SUBAPPLICATION SubApp_PC_B (* Geraet B (Station 12, 192.168.1.12): identisch zu Training_10 (2x AX_SUBSCRIBE_1 -> ILOCK_SWITCH_PROTECT_AX -> 2x logiBUS_QXA), zusaetzlich schreibt der tatsaechlich erreichte Zustand (UP_OUT/DOWN_OUT NACH Arbitrierung/Schutzzeit) per AX_SPLIT_2 + AX_CLIENT_1_0 zurueck an Geraet A fuer die GreenWhiteBackground-Anzeige - analog zum Vorbild SoftKeySR_PC_A_OPC.SUB (dort State-Write von B nach A, hier gleiches Prinzip). *)
  (* Standard: 61499-2; Description: Copyright (c) 2026 Meisterschulen am Ostbahnhof This program and the accompanying materials are made available under the terms of the Eclipse Public License 2.0 which is available at https://www.eclipse.org/legal/epl-2.0/ SPDX-License-Identifier: EPL-2.0 *)
  (* Version 1.0, 2026-09-05, Franz Höpfinger, Meisterschulen am Ostbahnhof, initial API and implementation and/or initial documentation *)
  PACKAGE subapp::Training_11_OPC_UA_RES;
  IMPORT VV::const::OPC_UA::myOpcUaAddresses::SW1_UP_LOCAL_READ;
  IMPORT VV::const::OPC_UA::myOpcUaAddresses::SW1_DOWN_LOCAL_READ;
  IMPORT VV::const::OPC_UA::myOpcUaAddresses::SW1_UP_STATE_REMOTE_WRITE;
  IMPORT VV::const::OPC_UA::myOpcUaAddresses::SW1_DOWN_STATE_REMOTE_WRITE;
  IMPORT logiBUS::io::DQ::logiBUS_DO::Output_Q7;
  IMPORT logiBUS::io::DQ::logiBUS_DO::Output_Q8;
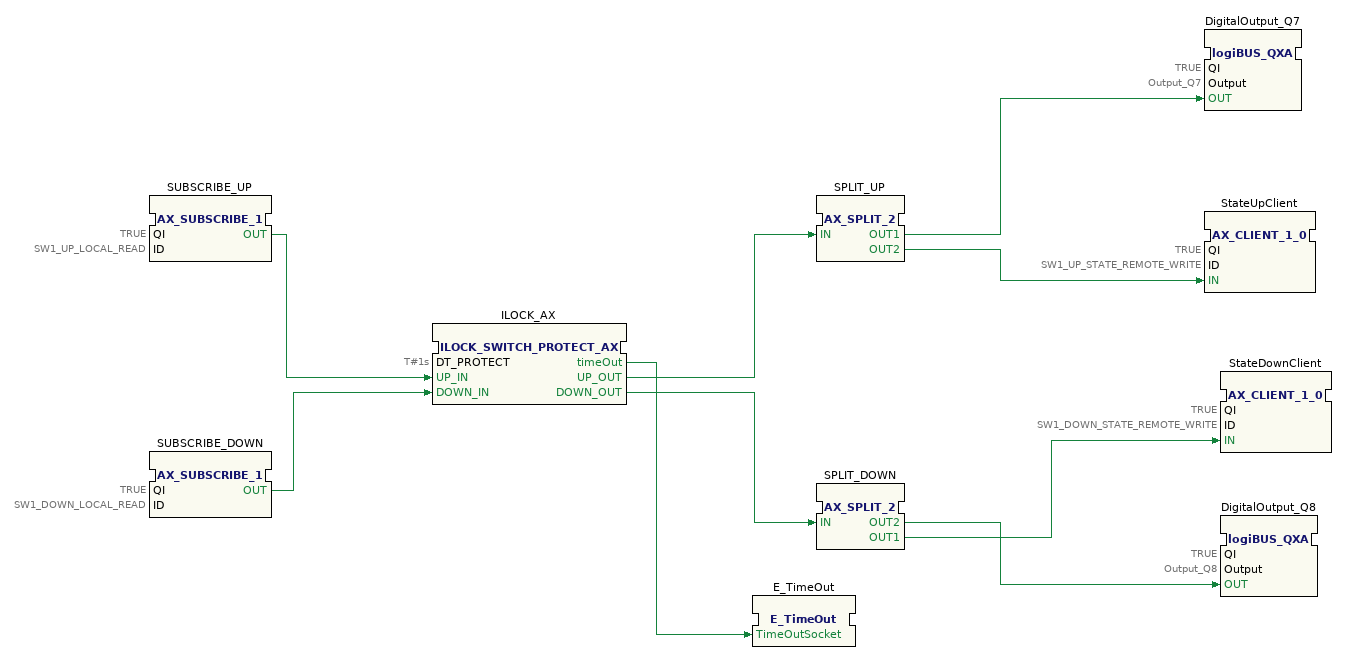
  FBS
    SUBSCRIBE_UP : adapter::net::AX_SUBSCRIBE_1(QI := TRUE, ID := SW1_UP_LOCAL_READ);
    SUBSCRIBE_DOWN : adapter::net::AX_SUBSCRIBE_1(QI := TRUE, ID := SW1_DOWN_LOCAL_READ);
    ILOCK_AX : logiBUS::signalprocessing::interlock::ILOCK_SWITCH_PROTECT_AX(DT_PROTECT := T#1s);
    E_TimeOut : iec61499::events::E_TimeOut;
    SPLIT_UP : adapter::events::unidirectional::AX_SPLIT_2;
    SPLIT_DOWN : adapter::events::unidirectional::AX_SPLIT_2;
    DigitalOutput_Q7 : logiBUS::io::DQ::logiBUS_QXA(QI := TRUE, Output := Output_Q7);
    DigitalOutput_Q8 : logiBUS::io::DQ::logiBUS_QXA(QI := TRUE, Output := Output_Q8);
    StateUpClient : adapter::net::AX_CLIENT_1_0(QI := TRUE, ID := SW1_UP_STATE_REMOTE_WRITE);
    StateDownClient : adapter::net::AX_CLIENT_1_0(QI := TRUE, ID := SW1_DOWN_STATE_REMOTE_WRITE);
  END_FBS
  ADAPTER_CONNECTIONS
    SUBSCRIBE_UP.OUT TO ILOCK_AX.UP_IN;
    SUBSCRIBE_DOWN.OUT TO ILOCK_AX.DOWN_IN;
    ILOCK_AX.timeOut TO E_TimeOut.TimeOutSocket;
    ILOCK_AX.UP_OUT TO SPLIT_UP.IN;
    SPLIT_UP.OUT1 TO DigitalOutput_Q7.OUT;
    SPLIT_UP.OUT2 TO StateUpClient.IN;
    ILOCK_AX.DOWN_OUT TO SPLIT_DOWN.IN;
    SPLIT_DOWN.OUT2 TO DigitalOutput_Q8.OUT;
    SPLIT_DOWN.OUT1 TO StateDownClient.IN;
  END_CONNECTIONS
END_SUBAPPLICATION
